# EPICS substitutions: ecmcApp/Db/SlitX-master-extra.substitutions
file "ecmc-extra.template"
{
pattern
{P,      M,      R,         PORT,    ADDR, PREC, HOMEPROC}
{IOC2:,  master, master-,   MCU1,    5,    3,    3}
}
